// TIA Portal V17 export
// export: Created 2025-03-05T08:01:23.0971358Z, ExportSetting WithDefaults, DisplayName Totally Integrated Automation Portal, DisplayVersion V17 Update 8, DisplayName TIA Portal Openness, DisplayVersion V17 Update 8, DisplayName TIA Portal Version Control Interface, DisplayVersion V17, DisplayName SINAMICS Startdrive Advanced, DisplayVersion V17 SP2, DisplayName SINAMICS Startdrive G110M, G120, G120C, G120D, G120P, G115D, DisplayVersion V17 SP2, DisplayName SINAMICS Startdrive G130, G150, S120, S150, SINAMICS MV, S210, DisplayVersion V17 SP2, DisplayName STEP 7 Professional, DisplayVersion V17 Update 8, DisplayName SINUMERIK ONE STEP 7 Toolbox, DisplayVersion V17 Update 12, DisplayName SINUMERIK 840D sl STEP 7 Toolbox, DisplayVersion V17 Update 12, DisplayName STEP 7 Safety, DisplayVersion V17 Update 6, DisplayName WinCC Advanced, DisplayVersion V17 Update 8
DATA_BLOCK "DB20220_TRUMPF_LASER_UNIT_01_POINTER"   // DB20220
{ DB_Accessible_From_OPC_UA := 'FALSE' }
VERSION : 0.1
// stored: AutoNumber false, DBAccessibleFromOPCUA false, DBAccessibleFromWebserver true, InstanceOfName FB20201_TRUMPF_GUIDE, InstanceOfType FB
"FB20201_TRUMPF_GUIDE"
   // VAR_INPUT
   //    iEXTERNAL_CONTROL_READY : Bool;
   //    iLASER_ACTIVE_ON : Bool;
   //    iMANUAL_START_REQUEST : Bool;
   //    iAUTO_START_REQUEST : Bool;
   //    "iMANUAL STOP REQUEST" : Bool;
   //    "iAUTO STOP REQUEST" : Bool;
   //    iMACHINE_ON_DELAYED : Bool;
   //    iSAFETY_GATES_CLOSED_LOCKED : Bool;
   //    iPILOT_LASER_IS_ON : Bool;
   // END_VAR
   // VAR_OUTPUT
   //    oGUIDE_SWITCH_ON : Bool;
   //    oLASER_POINTER_NOT_READY_ALARM : Bool;
   //    oSTATION_SEOC_ALARMS : Bool;
   //    oSwitchoncondition_off : Bool;
   //    oSwitchoncondition_on : Bool;
   //    oLimit_right : Bool;
   //    oLimit_left : Bool;
   // END_VAR
   // VAR RETAIN
   //    DATA : "LASER POINTER";
   //    "TIMER FAULT" { S7_SetPoint := 'True'} : TON_TIME;
   // END_VAR
BEGIN
END_DATA_BLOCK
